(* IEC 61131-3 sources: sphere-usecases/water-treatment/implementations/openplc/projects/controller_project, 4 files *)

(* ---- controller_clean.st ---- *)
TYPE
  HMI_UDT : STRUCT
    Start_PB : BOOL;
    Stop_PB : BOOL;
    Start_Active : BOOL;
    Stop_Active : BOOL;
  END_STRUCT;
  P1_UDT : STRUCT
    RW_Tank_tnk_lvl : REAL;
    RW_Pump_flow : REAL;
    RW_Tank_PR_Valve_sts : BOOL;
    RW_Tank_P6B_Valve_sts : BOOL;
    RW_Tank_P_Valve_sts : BOOL;
    RW_Pump_sts : BOOL;
    RW_Pump_fault : BOOL;
    RW_Pump : REAL;
    RW_Tank_PR_Valve : BOOL;
    RW_Tank_P_Valve : BOOL;
    RW_Pump_start : BOOL;
    RW_Pump_stop : BOOL;
    RW_Tank_P6B_Valve : BOOL;
  END_STRUCT;
  P2_UDT : STRUCT
    ChemTreat_NaCl_Tank_tnk_lvl : REAL;
    ChemTreat_NaOCl_Tank_tnk_lvl : REAL;
    ChemTreat_HCl_Tank_tnk_lvl : REAL;
    ChemTreat_NaCl_Tank_Valve_sts : BOOL;
    ChemTreat_NaOCl_Tank_Valve_sts : BOOL;
    ChemTreat_HCl_Tank_Valve_sts : BOOL;
    ChemTreat_NaCl_Tank_Valve : BOOL;
    ChemTreat_NaOCl_Tank_Valve : BOOL;
    ChemTreat_HCl_Tank_Valve : BOOL;
  END_STRUCT;
  P3_UDT : STRUCT
    Ultrafiltration_UFFT_Tank_tnk_lvl : REAL;
    Ultrafiltration_UFFT_Tank_Valve_sts : BOOL;
    Ultrafiltration_UF_Drain_Valve_sts : BOOL;
    Ultrafiltration_UF_ROFT_Valve_sts : BOOL;
    Ultrafiltration_UF_BWP_Valve_sts : BOOL;
    Ultrafiltration_UFFT_Tank_Valve : BOOL;
    Ultrafiltration_UF_Drain_Valve : BOOL;
    Ultrafiltration_UF_ROFT_Valve : BOOL;
    Ultrafiltration_UF_BWP_Valve : BOOL;
  END_STRUCT;
  Phases_UDT : STRUCT
    Filling : BOOL;
    Draining : BOOL;
  END_STRUCT;
  RW_tank_AL_UDT : STRUCT
    LL_alarm : BOOL;
    L_alarm : BOOL;
    H_alarm : BOOL;
    HH_alarm : BOOL;
  END_STRUCT;
  System_State_UDT : STRUCT
    IDLE : BOOL;
    START : BOOL;
    RUNNING : BOOL;
    SHUTDOWN : BOOL;
    Permissives : ARRAY [0..31] OF BOOL;
    Permissives_Ready : BOOL;
  END_STRUCT;
  SYS_MESSAGES : STRUCT
    ProgramScanTime : DINT;
    AvailableMemory : REAL;
    ControllerStatus : SINT;
    ScanTime : REAL;
  END_STRUCT;
END_TYPE

PROGRAM MainProgram
  VAR_INPUT
    Alarms : RW_tank_AL_UDT;
    GSV_Message : SYS_MESSAGES;
    P1 : P1_UDT;
    P1_SYS : System_State_UDT;
    P2 : P2_UDT;
    P3 : P3_UDT;
  END_VAR
  VAR_INPUT
    di_2_0 AT %IX2.0 : BOOL;
    di_2_1 AT %IX2.1 : BOOL;
    di_2_10 AT %IX2.10 : BOOL;
    di_2_11 AT %IX2.11 : BOOL;
    di_2_2 AT %IX2.2 : BOOL;
    di_2_3 AT %IX2.3 : BOOL;
    di_2_4 AT %IX2.4 : BOOL;
    di_2_5 AT %IX2.5 : BOOL;
    di_2_6 AT %IX2.6 : BOOL;
    di_2_8 AT %IX2.8 : BOOL;
    di_2_9 AT %IX2.9 : BOOL;
    ai_7_0 AT %IW70 : REAL;
    di_7_ch0halarm AT %IX7.0 : BOOL;
    di_7_ch0hhalarm AT %IX7.0 : BOOL;
    di_7_ch0lalarm AT %IX7.0 : BOOL;
    di_7_ch0llalarm AT %IX7.0 : BOOL;
    ai_7_1 AT %IW71 : REAL;
    ai_7_2 AT %IW72 : REAL;
    ai_7_3 AT %IW73 : REAL;
    ai_7_4 AT %IW74 : REAL;
    ai_7_5 AT %IW75 : REAL;
  END_VAR
  VAR_OUTPUT
    HMI : HMI_UDT;
  END_VAR
  VAR_OUTPUT
    ao_10_0 AT %QW100 : REAL;
    do_5_0 AT %QX5.0 : BOOL;
    do_5_1 AT %QX5.1 : BOOL;
    do_5_10 AT %QX5.10 : BOOL;
    do_5_11 AT %QX5.11 : BOOL;
    do_5_2 AT %QX5.2 : BOOL;
    do_5_3 AT %QX5.3 : BOOL;
    do_5_4 AT %QX5.4 : BOOL;
    do_5_5 AT %QX5.5 : BOOL;
    do_5_6 AT %QX5.6 : BOOL;
    do_5_7 AT %QX5.7 : BOOL;
    do_5_8 AT %QX5.8 : BOOL;
    do_5_9 AT %QX5.9 : BOOL;
  END_VAR

  (* IO_setup *)
  (* P1 Analog Input *)
  P1.RW_Tank_tnk_lvl := ai_7_0;
  P1.RW_Pump_flow := ai_7_1;
  (* P1 Digital Input *)
  P1.RW_Tank_PR_Valve_sts := di_2_0;
  P1.RW_Tank_P6B_Valve_sts := di_2_1;
  P1.RW_Tank_P_Valve_sts := di_2_2;
  P1.RW_Pump_sts := di_2_3;
  P1.RW_Pump_fault := di_2_4;
  (* P1 Analog Output *)
  P1.RW_Pump := ao_10_0;
  (* Digital Output *)
  P1.RW_Tank_PR_Valve := do_5_0;
  P1.RW_Tank_P6B_Valve := do_5_1;
  P1.RW_Tank_P_Valve := do_5_2;
  P1.RW_Pump_start := do_5_3;
  P1.RW_Pump_stop := do_5_4;
  (* P1 raw water tank alarms *)
  Alarms.LL_alarm := di_7_ch0llalarm;
  Alarms.L_alarm := di_7_ch0lalarm;
  Alarms.H_alarm := di_7_ch0halarm;
  Alarms.HH_alarm := di_7_ch0hhalarm;
  (* P2 Analog Input *)
  P2.ChemTreat_NaCl_Tank_tnk_lvl := ai_7_2;
  P2.ChemTreat_NaOCl_Tank_tnk_lvl := ai_7_3;
  P2.ChemTreat_HCl_Tank_tnk_lvl := ai_7_4;
  (* P2 Digital Input *)
  P2.ChemTreat_NaCl_Tank_Valve_sts := di_2_5;
  P2.ChemTreat_NaOCl_Tank_Valve_sts := di_2_6;
  (* P2 Analog Output *)
  (* NONE *)
  (* P2 Digital Output *)
  P2.ChemTreat_NaCl_Tank_Valve := do_5_5;
  P2.ChemTreat_NaOCl_Tank_Valve := do_5_6;
  P2.ChemTreat_HCl_Tank_Valve := do_5_7;
  (* P3 Analog Input *)
  P3.Ultrafiltration_UFFT_Tank_tnk_lvl := ai_7_5;
  (* P3 Digital Input *)
  P3.Ultrafiltration_UFFT_Tank_Valve_sts := di_2_8;
  P3.Ultrafiltration_UF_Drain_Valve_sts := di_2_9;
  P3.Ultrafiltration_UF_Drain_Valve_sts := di_2_10;
  P3.Ultrafiltration_UF_BWP_Valve_sts := di_2_11;
  (* P3 Analog Output *)
  (* none *)
  (* P3 Digital Output *)
  P3.Ultrafiltration_UFFT_Tank_Valve := do_5_8;
  P3.Ultrafiltration_UF_Drain_Valve := do_5_9;
  P3.Ultrafiltration_UF_ROFT_Valve := do_5_10;
  P3.Ultrafiltration_UF_BWP_Valve := do_5_11;

  (* Raw_water_control *)
  if P1.RW_Tank_tnk_lvl = 250.0 and P1_SYS.RUNNING then
  P1.RW_Pump_stop := True;
  P1.RW_Pump_start := False; (* send the outputs *)
  Alarms.LL_alarm := True;
  (* if the level is at 500 or lower than 500 open the valve *)
  elsif P1.RW_Tank_tnk_lvl <= 500.0 and P1_SYS.RUNNING then
  (* output to turn the valve open *)
  P1.RW_Tank_PR_Valve := True;
  Alarms.L_alarm := True;
  (* if level is at 800 *)
  elsif  P1.RW_Tank_tnk_lvl = 800.0 and P1_SYS.RUNNING then
  P1.RW_Tank_PR_Valve := False; (* close the valve *)
  Alarms.H_alarm := True;
  elsif P1.RW_Tank_tnk_lvl = 1200.0 and P1_SYS.RUNNING then
  Alarms.HH_alarm := True; (* if the tank is higher than or equal to 1200 set the high high alarm *)
  end_if;

  (* Raw_water_pump *)
  if P3.Ultrafiltration_UFFT_Tank_tnk_lvl = 800.0 AND P1_SYS.RUNNING then
  (* start the pump and open the valve from the other tank *)
  P1.RW_Tank_P_Valve := True;
  P1.RW_Pump_start := True;
  P1.RW_Pump_stop := False;
  elsif P3.Ultrafiltration_UFFT_Tank_tnk_lvl = 1000.0 AND P1_SYS.RUNNING then
  (* stop the pump and close the valve *)
  P1.RW_Tank_P_Valve := False;
  P1.RW_Pump_stop := True;
  P1.RW_Pump_start := False;
  end_if;

  (* State_change *)
  if not HMI.Start_Active AND not HMI.Stop_Active then
  (* if start and stop is not pressed go to idle *)
  P1_SYS.IDLE := True;
  P1_SYS.START := False;
  P1_SYS.RUNNING := False;
  P1_SYS.SHUTDOWN := False;
  elsif  HMI.Start_Active AND not HMI.Stop_Active then
  (* if the start pb and stop is not pressed then change the state of process one to starting *)
  P1_SYS.IDLE := False;
  P1_SYS.START := True;
  P1_SYS.RUNNING := False;
  P1_SYS.SHUTDOWN := False;
  (* if the tank level is greater than 250 at the start and UFFT is less than a 1000 we can start *)
  (* then and all permissves cond together into one tag so we know the plant is ready to start *)
  P1_SYS.Permissives_Ready := P1_SYS.Permissives[0] AND P1_SYS.Permissives[1];
  elsif HMI.Start_Active AND P1_SYS.Permissives_Ready then
  (* if the start was pressed and permissives are ready start running Process one *)
  P1_SYS.IDLE := False;
  P1_SYS.START := False;
  P1_SYS.RUNNING := True;
  P1_SYS.SHUTDOWN := False;
  elsif HMI.Stop_Active then
  (* if the stop button is pressed then go to shutdown state *)
  P1_SYS.IDLE := False;
  P1_SYS.START := False;
  P1_SYS.RUNNING := False;
  P1_SYS.SHUTDOWN := True;
  (* set all permissives to false *)
  P1_SYS.Permissives_Ready := False;
  end_if;
END_PROGRAM

CONFIGURATION config
  VAR_GLOBAL
    ao_10_0 AT %QW100 : REAL;
    di_2_0 AT %IX2.0 : BOOL;
    di_2_1 AT %IX2.1 : BOOL;
    di_2_10 AT %IX2.10 : BOOL;
    di_2_11 AT %IX2.11 : BOOL;
    di_2_2 AT %IX2.2 : BOOL;
    di_2_3 AT %IX2.3 : BOOL;
    di_2_4 AT %IX2.4 : BOOL;
    di_2_5 AT %IX2.5 : BOOL;
    di_2_6 AT %IX2.6 : BOOL;
    di_2_8 AT %IX2.8 : BOOL;
    di_2_9 AT %IX2.9 : BOOL;
    do_5_0 AT %QX5.0 : BOOL;
    do_5_1 AT %QX5.1 : BOOL;
    do_5_10 AT %QX5.10 : BOOL;
    do_5_11 AT %QX5.11 : BOOL;
    do_5_2 AT %QX5.2 : BOOL;
    do_5_3 AT %QX5.3 : BOOL;
    do_5_4 AT %QX5.4 : BOOL;
    do_5_5 AT %QX5.5 : BOOL;
    do_5_6 AT %QX5.6 : BOOL;
    do_5_7 AT %QX5.7 : BOOL;
    do_5_8 AT %QX5.8 : BOOL;
    do_5_9 AT %QX5.9 : BOOL;
    ai_7_0 AT %IW70 : REAL;
    di_7_ch0halarm AT %IX7.0 : BOOL;
    di_7_ch0hhalarm AT %IX7.0 : BOOL;
    di_7_ch0lalarm AT %IX7.0 : BOOL;
    di_7_ch0llalarm AT %IX7.0 : BOOL;
    ai_7_1 AT %IW71 : REAL;
    ai_7_2 AT %IW72 : REAL;
    ai_7_3 AT %IW73 : REAL;
    ai_7_4 AT %IW74 : REAL;
    ai_7_5 AT %IW75 : REAL;
  END_VAR

  RESOURCE res_MainProgram ON PLC
    TASK task_MainProgram(INTERVAL := T#100ms,PRIORITY := 0);
    PROGRAM MainProgram_instance : MainProgram;
  END_RESOURCE
END_CONFIGURATION

(* ---- controller_final.st ---- *)
TYPE
  HMI_UDT : STRUCT
    Start_PB : BOOL;
    Stop_PB : BOOL;
    Reset_PB : BOOL;
    Start_Active : BOOL;
    Stop_Active : BOOL;
  END_STRUCT;
  P1_UDT : STRUCT
    RW_Tank_tnk_lvl : REAL;
    RW_Pump_flow : REAL;
    RW_Tank_PR_Valve_sts : BOOL;
    RW_Tank_P6B_Valve_sts : BOOL;
    RW_Tank_P_Valve_sts : BOOL;
    RW_Pump_sts : BOOL;
    RW_Pump_fault : BOOL;
    RW_Pump : REAL;
    RW_Tank_PR_Valve : BOOL;
    RW_Tank_P_Valve : BOOL;
    RW_Pump_start : BOOL;
    RW_Pump_stop : BOOL;
    RW_Tank_P6B_Valve : BOOL;
  END_STRUCT;
  P2_UDT : STRUCT
    ChemTreat_NaCl_Tank_tnk_lvl : REAL;
    ChemTreat_NaOCl_Tank_tnk_lvl : REAL;
    ChemTreat_HCl_Tank_tnk_lvl : REAL;
    ChemTreat_NaCl_Tank_Valve_sts : BOOL;
    ChemTreat_NaOCl_Tank_Valve_sts : BOOL;
    ChemTreat_HCl_Tank_Valve_sts : BOOL;
    ChemTreat_NaCl_Tank_Valve : BOOL;
    ChemTreat_NaOCl_Tank_Valve : BOOL;
    ChemTreat_HCl_Tank_Valve : BOOL;
  END_STRUCT;
  P3_UDT : STRUCT
    Ultrafiltration_UFFT_Tank_tnk_lvl : REAL;
    Ultrafiltration_UFFT_Tank_Valve_sts : BOOL;
    Ultrafiltration_UF_Drain_Valve_sts : BOOL;
    Ultrafiltration_UF_ROFT_Valve_sts : BOOL;
    Ultrafiltration_UF_BWP_Valve_sts : BOOL;
    Ultrafiltration_UFFT_Tank_Valve : BOOL;
    Ultrafiltration_UF_Drain_Valve : BOOL;
    Ultrafiltration_UF_ROFT_Valve : BOOL;
    Ultrafiltration_UF_BWP_Valve : BOOL;
  END_STRUCT;
  Phases_UDT : STRUCT
    Filling : BOOL;
    Draining : BOOL;
  END_STRUCT;
  RW_tank_AL_UDT : STRUCT
    LL_alarm : BOOL;
    L_alarm : BOOL;
    H_alarm : BOOL;
    HH_alarm : BOOL;
  END_STRUCT;
  System_State_UDT : STRUCT
    IDLE : BOOL;
    START : BOOL;
    RUNNING : BOOL;
    SHUTDOWN : BOOL;
    Permissives : ARRAY [0..31] OF BOOL;
    Permissives_Ready : BOOL;
  END_STRUCT;
  SYS_MESSAGES : STRUCT
    ProgramScanTime : DINT;
    AvailableMemory : REAL;
    ControllerStatus : SINT;
    ScanTime : REAL;
  END_STRUCT;
END_TYPE

PROGRAM MainProgram
  VAR
    HMI : HMI_UDT;
    Alarms : RW_tank_AL_UDT;
    GSV_Message : SYS_MESSAGES;
    Init_Done : BOOL := FALSE;
    P1 : P1_UDT;
    P1_SYS : System_State_UDT;
    P2 : P2_UDT;
    P3 : P3_UDT;
  END_VAR
  VAR_EXTERNAL
    ao_10_0 : INT;
    do_5_0 : BOOL;
    do_5_1 : BOOL;
    do_5_10 : BOOL;
    do_5_11 : BOOL;
    do_5_2 : BOOL;
    do_5_3 : BOOL;
    do_5_4 : BOOL;
    do_5_5 : BOOL;
    do_5_6 : BOOL;
    do_5_7 : BOOL;
    do_5_8 : BOOL;
    do_5_9 : BOOL;
    (* HMI coils %QX0.0-0.3 *)
    hmi_0_0 : BOOL;  (* HMI_Start_PB - written by external client *)
    hmi_0_1 : BOOL;  (* HMI_Stop_PB  - written by external client *)
    hmi_0_2 : BOOL;  (* HMI_Start_Active - written by controller *)
    hmi_0_3 : BOOL;  (* HMI_Stop_Active  - written by controller *)
    hmi_0_4 : BOOL;  (* HMI_Reset_PB - written by external client *)
    (* Process selection/manual P2 control coils %QX1.0-1.3 *)
    p2_1_0 : BOOL;  (* P2_Selected - written by external client *)
    p2_1_1 : BOOL;  (* P2_NaCl_Cmd - written by external client *)
    p2_1_2 : BOOL;  (* P2_NaOCl_Cmd - written by external client *)
    p2_1_3 : BOOL;  (* P2_HCl_Cmd - written by external client *)
    (* System state coils %QX7.0-7.4 *)
    sys_7_0 : BOOL;  (* SYS_IDLE *)
    sys_7_1 : BOOL;  (* SYS_START *)
    sys_7_2 : BOOL;  (* SYS_RUNNING *)
    sys_7_3 : BOOL;  (* SYS_SHUTDOWN *)
    sys_7_4 : BOOL;  (* SYS_Permissives_Ready *)
    (* Alarm coils %QX8.0-8.3 *)
    alm_8_0 : BOOL;  (* Alarm_RW_Tank_LL *)
    alm_8_1 : BOOL;  (* Alarm_RW_Tank_L *)
    alm_8_2 : BOOL;  (* Alarm_RW_Tank_H *)
    alm_8_3 : BOOL;  (* Alarm_RW_Tank_HH *)
    (* Bridge sensor inputs - holding registers written by bridge *)
    bridge_rw_level : INT;       (* %QW300 - RW tank level from simulator *)
    bridge_rw_flow : INT;        (* %QW301 - RW pump flow from simulator *)
    bridge_nacl_level : INT;     (* %QW302 - NaCl tank level *)
    bridge_naocl_level : INT;    (* %QW303 - NaOCl tank level *)
    bridge_hcl_level : INT;      (* %QW304 - HCl tank level *)
    bridge_uf_level : INT;       (* %QW305 - UF tank level *)
    bridge_pr_valve_sts : INT;   (* %QW320 - PR valve status *)
    bridge_p6b_valve_sts : INT;  (* %QW321 - P6B valve status *)
    bridge_p_valve_sts : INT;    (* %QW322 - P valve status *)
    bridge_pump_sts : INT;       (* %QW323 - pump running status *)
    bridge_pump_fault : INT;     (* %QW324 - pump fault *)
    bridge_nacl_valve_sts : INT; (* %QW325 - NaCl valve status *)
    bridge_naocl_valve_sts : INT;(* %QW326 - NaOCl valve status *)
    bridge_hcl_valve_sts : INT;  (* %QW327 - HCl valve status *)
    bridge_uf_valve_sts : INT;   (* %QW328 - UF tank valve status *)
    bridge_uf_drain_sts : INT;   (* %QW329 - UF drain valve status *)
    bridge_uf_roft_sts : INT;    (* %QW330 - UF ROFT valve status *)
    bridge_uf_bwp_sts : INT;     (* %QW331 - UF BWP valve status *)
  END_VAR

  IF NOT Init_Done THEN
    HMI.Start_Active := FALSE;
    HMI.Stop_Active := FALSE;
    P1_SYS.IDLE := TRUE;
    P1_SYS.START := FALSE;
    P1_SYS.RUNNING := FALSE;
    P1_SYS.SHUTDOWN := FALSE;
    P1_SYS.Permissives_Ready := FALSE;
    P1.RW_Pump := 0.0;
    P1.RW_Tank_PR_Valve := FALSE;
    P1.RW_Tank_P_Valve := FALSE;
    P1.RW_Pump_start := FALSE;
    P1.RW_Pump_stop := TRUE;
    P1.RW_Tank_P6B_Valve := FALSE;
    P2.ChemTreat_NaCl_Tank_Valve := FALSE;
    P2.ChemTreat_NaOCl_Tank_Valve := FALSE;
    P2.ChemTreat_HCl_Tank_Valve := FALSE;
    P3.Ultrafiltration_UFFT_Tank_Valve := FALSE;
    P3.Ultrafiltration_UF_Drain_Valve := FALSE;
    P3.Ultrafiltration_UF_ROFT_Valve := FALSE;
    P3.Ultrafiltration_UF_BWP_Valve := FALSE;
    Init_Done := TRUE;
  END_IF;

  (* ===== HMI button latch ===== *)
  HMI.Start_PB := hmi_0_0;
  HMI.Stop_PB := hmi_0_1;
  HMI.Reset_PB := hmi_0_4;
  IF HMI.Reset_PB THEN
    HMI.Start_Active := FALSE;
    HMI.Stop_Active := FALSE;
  ELSIF HMI.Start_PB THEN
    HMI.Start_Active := TRUE;
    HMI.Stop_Active := FALSE;
  ELSIF HMI.Stop_PB THEN
    HMI.Stop_Active := TRUE;
    HMI.Start_Active := FALSE;
  END_IF;

  (* ===== Read sensors from bridge holding registers ===== *)
  (* Levels: INT -> REAL conversion *)
  P1.RW_Tank_tnk_lvl := INT_TO_REAL(bridge_rw_level);
  P1.RW_Pump_flow := INT_TO_REAL(bridge_rw_flow);
  P2.ChemTreat_NaCl_Tank_tnk_lvl := INT_TO_REAL(bridge_nacl_level);
  P2.ChemTreat_NaOCl_Tank_tnk_lvl := INT_TO_REAL(bridge_naocl_level);
  P2.ChemTreat_HCl_Tank_tnk_lvl := INT_TO_REAL(bridge_hcl_level);
  P3.Ultrafiltration_UFFT_Tank_tnk_lvl := INT_TO_REAL(bridge_uf_level);
  (* Valve/pump status: INT -> BOOL (nonzero = TRUE) *)
  P1.RW_Tank_PR_Valve_sts := bridge_pr_valve_sts <> 0;
  P1.RW_Tank_P6B_Valve_sts := bridge_p6b_valve_sts <> 0;
  P1.RW_Tank_P_Valve_sts := bridge_p_valve_sts <> 0;
  P1.RW_Pump_sts := bridge_pump_sts <> 0;
  P1.RW_Pump_fault := bridge_pump_fault <> 0;
  P2.ChemTreat_NaCl_Tank_Valve_sts := bridge_nacl_valve_sts <> 0;
  P2.ChemTreat_NaOCl_Tank_Valve_sts := bridge_naocl_valve_sts <> 0;
  P3.Ultrafiltration_UFFT_Tank_Valve_sts := bridge_uf_valve_sts <> 0;
  P3.Ultrafiltration_UF_Drain_Valve_sts := bridge_uf_drain_sts <> 0;
  P3.Ultrafiltration_UF_ROFT_Valve_sts := bridge_uf_roft_sts <> 0;
  P3.Ultrafiltration_UF_BWP_Valve_sts := bridge_uf_bwp_sts <> 0;

  (* ===== Compute alarms from levels ===== *)
  Alarms.LL_alarm := P1.RW_Tank_tnk_lvl <= 250.0;
  Alarms.L_alarm := P1.RW_Tank_tnk_lvl <= 500.0;
  Alarms.H_alarm := P1.RW_Tank_tnk_lvl >= 800.0;
  Alarms.HH_alarm := P1.RW_Tank_tnk_lvl >= 1200.0;

  (* ===== Permissives ===== *)
  P1_SYS.Permissives[0] := P1.RW_Tank_tnk_lvl > 250.0;
  P1_SYS.Permissives[1] := P3.Ultrafiltration_UFFT_Tank_tnk_lvl < 1000.0;
  P1_SYS.Permissives_Ready := P1_SYS.Permissives[0] AND P1_SYS.Permissives[1];

  (* ===== State_change ===== *)
  IF HMI.Reset_PB THEN
    P1_SYS.IDLE := TRUE;
    P1_SYS.START := FALSE;
    P1_SYS.RUNNING := FALSE;
    P1_SYS.SHUTDOWN := FALSE;
    P1_SYS.Permissives_Ready := FALSE;
    P1.RW_Pump := 0.0;
    P1.RW_Tank_PR_Valve := FALSE;
    P1.RW_Tank_P_Valve := FALSE;
    P1.RW_Pump_start := FALSE;
    P1.RW_Pump_stop := TRUE;
  ELSIF NOT HMI.Start_Active AND NOT HMI.Stop_Active THEN
    P1_SYS.IDLE := TRUE;
    P1_SYS.START := FALSE;
    P1_SYS.RUNNING := FALSE;
    P1_SYS.SHUTDOWN := FALSE;
    P1_SYS.Permissives_Ready := FALSE;
    P1.RW_Pump := 0.0;
    P1.RW_Tank_PR_Valve := FALSE;
    P1.RW_Tank_P_Valve := FALSE;
    P1.RW_Pump_start := FALSE;
    P1.RW_Pump_stop := TRUE;
  ELSIF HMI.Start_Active AND NOT HMI.Stop_Active AND NOT P1_SYS.Permissives_Ready THEN
    P1_SYS.IDLE := FALSE;
    P1_SYS.START := TRUE;
    P1_SYS.RUNNING := FALSE;
    P1_SYS.SHUTDOWN := FALSE;
  ELSIF HMI.Start_Active AND P1_SYS.Permissives_Ready THEN
    P1_SYS.IDLE := FALSE;
    P1_SYS.START := FALSE;
    P1_SYS.RUNNING := TRUE;
    P1_SYS.SHUTDOWN := FALSE;
  ELSIF HMI.Stop_Active THEN
    P1_SYS.IDLE := FALSE;
    P1_SYS.START := FALSE;
    P1_SYS.RUNNING := FALSE;
    P1_SYS.SHUTDOWN := TRUE;
    P1_SYS.Permissives_Ready := FALSE;
    P1.RW_Pump := 0.0;
    P1.RW_Tank_PR_Valve := FALSE;
    P1.RW_Tank_P_Valve := FALSE;
    P1.RW_Pump_start := FALSE;
    P1.RW_Pump_stop := TRUE;
  END_IF;

  (* ===== Raw_water_control ===== *)
  IF P1_SYS.RUNNING THEN
    IF P1.RW_Tank_tnk_lvl <= 250.0 THEN
      P1.RW_Pump_stop := TRUE;
      P1.RW_Pump_start := FALSE;
      P1.RW_Tank_P_Valve := FALSE;
      P1.RW_Pump := 0.0;
    ELSIF P1.RW_Tank_tnk_lvl <= 500.0 THEN
      P1.RW_Tank_PR_Valve := TRUE;
    ELSIF P1.RW_Tank_tnk_lvl >= 800.0 THEN
      P1.RW_Tank_PR_Valve := FALSE;
    END_IF;

    (* ===== Raw_water_pump ===== *)
    IF P3.Ultrafiltration_UFFT_Tank_tnk_lvl <= 800.0 THEN
      P1.RW_Tank_P_Valve := TRUE;
      P1.RW_Pump_start := TRUE;
      P1.RW_Pump_stop := FALSE;
      P1.RW_Pump := 100.0;
    ELSIF P3.Ultrafiltration_UFFT_Tank_tnk_lvl >= 1000.0 THEN
      P1.RW_Tank_P_Valve := FALSE;
      P1.RW_Pump_stop := TRUE;
      P1.RW_Pump_start := FALSE;
      P1.RW_Pump := 0.0;
    END_IF;
  END_IF;

  (* ===== Manual Process 2 control ===== *)
  IF P1_SYS.RUNNING AND p2_1_0 THEN
    P2.ChemTreat_NaCl_Tank_Valve := p2_1_1;
    P2.ChemTreat_NaOCl_Tank_Valve := p2_1_2;
    P2.ChemTreat_HCl_Tank_Valve := p2_1_3;
  ELSE
    P2.ChemTreat_NaCl_Tank_Valve := FALSE;
    P2.ChemTreat_NaOCl_Tank_Valve := FALSE;
    P2.ChemTreat_HCl_Tank_Valve := FALSE;
  END_IF;

  (* ===== Wire outputs to coils/registers ===== *)
  do_5_0 := P1.RW_Tank_PR_Valve;
  do_5_1 := P1.RW_Tank_P6B_Valve;
  do_5_2 := P1.RW_Tank_P_Valve;
  do_5_3 := P1.RW_Pump_start;
  do_5_4 := P1.RW_Pump_stop;
  do_5_5 := P2.ChemTreat_NaCl_Tank_Valve;
  do_5_6 := P2.ChemTreat_NaOCl_Tank_Valve;
  do_5_7 := P2.ChemTreat_HCl_Tank_Valve;
  do_5_8 := P3.Ultrafiltration_UFFT_Tank_Valve;
  do_5_9 := P3.Ultrafiltration_UF_Drain_Valve;
  do_5_10 := P3.Ultrafiltration_UF_ROFT_Valve;
  do_5_11 := P3.Ultrafiltration_UF_BWP_Valve;
  ao_10_0 := REAL_TO_INT(P1.RW_Pump);
  (* HMI status *)
  hmi_0_2 := HMI.Start_Active;
  hmi_0_3 := HMI.Stop_Active;
  (* System state *)
  sys_7_0 := P1_SYS.IDLE;
  sys_7_1 := P1_SYS.START;
  sys_7_2 := P1_SYS.RUNNING;
  sys_7_3 := P1_SYS.SHUTDOWN;
  sys_7_4 := P1_SYS.Permissives_Ready;
  (* Alarms *)
  alm_8_0 := Alarms.LL_alarm;
  alm_8_1 := Alarms.L_alarm;
  alm_8_2 := Alarms.H_alarm;
  alm_8_3 := Alarms.HH_alarm;
END_PROGRAM

CONFIGURATION Config0
  VAR_GLOBAL
    ao_10_0 AT %QW100 : INT;
    do_5_0 AT %QX5.0 : BOOL;
    do_5_1 AT %QX5.1 : BOOL;
    do_5_10 AT %QX5.10 : BOOL;
    do_5_11 AT %QX5.11 : BOOL;
    do_5_2 AT %QX5.2 : BOOL;
    do_5_3 AT %QX5.3 : BOOL;
    do_5_4 AT %QX5.4 : BOOL;
    do_5_5 AT %QX5.5 : BOOL;
    do_5_6 AT %QX5.6 : BOOL;
    do_5_7 AT %QX5.7 : BOOL;
    do_5_8 AT %QX5.8 : BOOL;
    do_5_9 AT %QX5.9 : BOOL;
    (* HMI coils %QX0.0-0.4 *)
    hmi_0_0 AT %QX0.0 : BOOL;
    hmi_0_1 AT %QX0.1 : BOOL;
    hmi_0_2 AT %QX0.2 : BOOL;
    hmi_0_3 AT %QX0.3 : BOOL;
    hmi_0_4 AT %QX0.4 : BOOL;
    (* Process selection/manual P2 control coils %QX1.0-1.3 *)
    p2_1_0 AT %QX1.0 : BOOL;
    p2_1_1 AT %QX1.1 : BOOL;
    p2_1_2 AT %QX1.2 : BOOL;
    p2_1_3 AT %QX1.3 : BOOL;
    (* System state coils %QX7.0-7.4 *)
    sys_7_0 AT %QX7.0 : BOOL;
    sys_7_1 AT %QX7.1 : BOOL;
    sys_7_2 AT %QX7.2 : BOOL;
    sys_7_3 AT %QX7.3 : BOOL;
    sys_7_4 AT %QX7.4 : BOOL;
    (* Alarm coils %QX8.0-8.3 *)
    alm_8_0 AT %QX8.0 : BOOL;
    alm_8_1 AT %QX8.1 : BOOL;
    alm_8_2 AT %QX8.2 : BOOL;
    alm_8_3 AT %QX8.3 : BOOL;
    (* Bridge sensor inputs - holding registers writable by bridge *)
    bridge_rw_level AT %QW300 : INT;
    bridge_rw_flow AT %QW301 : INT;
    bridge_nacl_level AT %QW302 : INT;
    bridge_naocl_level AT %QW303 : INT;
    bridge_hcl_level AT %QW304 : INT;
    bridge_uf_level AT %QW305 : INT;
    bridge_pr_valve_sts AT %QW320 : INT;
    bridge_p6b_valve_sts AT %QW321 : INT;
    bridge_p_valve_sts AT %QW322 : INT;
    bridge_pump_sts AT %QW323 : INT;
    bridge_pump_fault AT %QW324 : INT;
    bridge_nacl_valve_sts AT %QW325 : INT;
    bridge_naocl_valve_sts AT %QW326 : INT;
    bridge_hcl_valve_sts AT %QW327 : INT;
    bridge_uf_valve_sts AT %QW328 : INT;
    bridge_uf_drain_sts AT %QW329 : INT;
    bridge_uf_roft_sts AT %QW330 : INT;
    bridge_uf_bwp_sts AT %QW331 : INT;
  END_VAR

  RESOURCE Res0 ON PLC
    TASK task_MainProgram(INTERVAL := T#100ms, PRIORITY := 0);
    PROGRAM MainProgram_instance : MainProgram;
  END_RESOURCE
END_CONFIGURATION

(* ---- controller_fixed.st ---- *)
TYPE
  HMI_UDT : STRUCT
    Start_PB : BOOL;
    Stop_PB : BOOL;
    Start_Active : BOOL;
    Stop_Active : BOOL;
  END_STRUCT;
  P1_UDT : STRUCT
    RW_Tank_tnk_lvl : REAL;
    RW_Pump_flow : REAL;
    RW_Tank_PR_Valve_sts : BOOL;
    RW_Tank_P6B_Valve_sts : BOOL;
    RW_Tank_P_Valve_sts : BOOL;
    RW_Pump_sts : BOOL;
    RW_Pump_fault : BOOL;
    RW_Pump : REAL;
    RW_Tank_PR_Valve : BOOL;
    RW_Tank_P_Valve : BOOL;
    RW_Pump_start : BOOL;
    RW_Pump_stop : BOOL;
    RW_Tank_P6B_Valve : BOOL;
  END_STRUCT;
  P2_UDT : STRUCT
    ChemTreat_NaCl_Tank_tnk_lvl : REAL;
    ChemTreat_NaOCl_Tank_tnk_lvl : REAL;
    ChemTreat_HCl_Tank_tnk_lvl : REAL;
    ChemTreat_NaCl_Tank_Valve_sts : BOOL;
    ChemTreat_NaOCl_Tank_Valve_sts : BOOL;
    ChemTreat_HCl_Tank_Valve_sts : BOOL;
    ChemTreat_NaCl_Tank_Valve : BOOL;
    ChemTreat_NaOCl_Tank_Valve : BOOL;
    ChemTreat_HCl_Tank_Valve : BOOL;
  END_STRUCT;
  P3_UDT : STRUCT
    Ultrafiltration_UFFT_Tank_tnk_lvl : REAL;
    Ultrafiltration_UFFT_Tank_Valve_sts : BOOL;
    Ultrafiltration_UF_Drain_Valve_sts : BOOL;
    Ultrafiltration_UF_ROFT_Valve_sts : BOOL;
    Ultrafiltration_UF_BWP_Valve_sts : BOOL;
    Ultrafiltration_UFFT_Tank_Valve : BOOL;
    Ultrafiltration_UF_Drain_Valve : BOOL;
    Ultrafiltration_UF_ROFT_Valve : BOOL;
    Ultrafiltration_UF_BWP_Valve : BOOL;
  END_STRUCT;
  Phases_UDT : STRUCT
    Filling : BOOL;
    Draining : BOOL;
  END_STRUCT;
  RW_tank_AL_UDT : STRUCT
    LL_alarm : BOOL;
    L_alarm : BOOL;
    H_alarm : BOOL;
    HH_alarm : BOOL;
  END_STRUCT;
  System_State_UDT : STRUCT
    IDLE : BOOL;
    START : BOOL;
    RUNNING : BOOL;
    SHUTDOWN : BOOL;
    Permissives : ARRAY [0..31] OF BOOL;
    Permissives_Ready : BOOL;
  END_STRUCT;
  SYS_MESSAGES : STRUCT
    ProgramScanTime : DINT;
    AvailableMemory : REAL;
    ControllerStatus : SINT;
    ScanTime : REAL;
  END_STRUCT;
END_TYPE

PROGRAM MainProgram
  VAR_INPUT
    Alarms : RW_tank_AL_UDT;
    GSV_Message : SYS_MESSAGES;
    P1 : P1_UDT;
    P1_SYS : System_State_UDT;
    P2 : P2_UDT;
    P3 : P3_UDT;
  END_VAR
  VAR_INPUT
    di_2_0 : BOOL;
    di_2_1 : BOOL;
    di_2_10 : BOOL;
    di_2_11 : BOOL;
    di_2_2 : BOOL;
    di_2_3 : BOOL;
    di_2_4 : BOOL;
    di_2_5 : BOOL;
    di_2_6 : BOOL;
    di_2_8 : BOOL;
    di_2_9 : BOOL;
    ai_7_0 : REAL;
    di_7_ch0halarm : BOOL;
    di_7_ch0hhalarm : BOOL;
    di_7_ch0lalarm : BOOL;
    di_7_ch0llalarm : BOOL;
    ai_7_1 : REAL;
    ai_7_2 : REAL;
    ai_7_3 : REAL;
    ai_7_4 : REAL;
    ai_7_5 : REAL;
  END_VAR
  VAR_OUTPUT
    HMI : HMI_UDT;
  END_VAR
  VAR_OUTPUT
    ao_10_0 : REAL;
    do_5_0 : BOOL;
    do_5_1 : BOOL;
    do_5_10 : BOOL;
    do_5_11 : BOOL;
    do_5_2 : BOOL;
    do_5_3 : BOOL;
    do_5_4 : BOOL;
    do_5_5 : BOOL;
    do_5_6 : BOOL;
    do_5_7 : BOOL;
    do_5_8 : BOOL;
    do_5_9 : BOOL;
  END_VAR

  (* IO_setup *)
  (* P1 Analog Input *)
  P1.RW_Tank_tnk_lvl := ai_7_0;
  P1.RW_Pump_flow := ai_7_1;
  (* P1 Digital Input *)
  P1.RW_Tank_PR_Valve_sts := di_2_0;
  P1.RW_Tank_P6B_Valve_sts := di_2_1;
  P1.RW_Tank_P_Valve_sts := di_2_2;
  P1.RW_Pump_sts := di_2_3;
  P1.RW_Pump_fault := di_2_4;
  (* P1 Analog Output *)
  P1.RW_Pump := ao_10_0;
  (* Digital Output *)
  P1.RW_Tank_PR_Valve := do_5_0;
  P1.RW_Tank_P6B_Valve := do_5_1;
  P1.RW_Tank_P_Valve := do_5_2;
  P1.RW_Pump_start := do_5_3;
  P1.RW_Pump_stop := do_5_4;
  (* P1 raw water tank alarms *)
  Alarms.LL_alarm := di_7_ch0llalarm;
  Alarms.L_alarm := di_7_ch0lalarm;
  Alarms.H_alarm := di_7_ch0halarm;
  Alarms.HH_alarm := di_7_ch0hhalarm;
  (* P2 Analog Input *)
  P2.ChemTreat_NaCl_Tank_tnk_lvl := ai_7_2;
  P2.ChemTreat_NaOCl_Tank_tnk_lvl := ai_7_3;
  P2.ChemTreat_HCl_Tank_tnk_lvl := ai_7_4;
  (* P2 Digital Input *)
  P2.ChemTreat_NaCl_Tank_Valve_sts := di_2_5;
  P2.ChemTreat_NaOCl_Tank_Valve_sts := di_2_6;
  (* P2 Analog Output *)
  (* NONE *)
  (* P2 Digital Output *)
  P2.ChemTreat_NaCl_Tank_Valve := do_5_5;
  P2.ChemTreat_NaOCl_Tank_Valve := do_5_6;
  P2.ChemTreat_HCl_Tank_Valve := do_5_7;
  (* P3 Analog Input *)
  P3.Ultrafiltration_UFFT_Tank_tnk_lvl := ai_7_5;
  (* P3 Digital Input *)
  P3.Ultrafiltration_UFFT_Tank_Valve_sts := di_2_8;
  P3.Ultrafiltration_UF_Drain_Valve_sts := di_2_9;
  P3.Ultrafiltration_UF_Drain_Valve_sts := di_2_10;
  P3.Ultrafiltration_UF_BWP_Valve_sts := di_2_11;
  (* P3 Analog Output *)
  (* none *)
  (* P3 Digital Output *)
  P3.Ultrafiltration_UFFT_Tank_Valve := do_5_8;
  P3.Ultrafiltration_UF_Drain_Valve := do_5_9;
  P3.Ultrafiltration_UF_ROFT_Valve := do_5_10;
  P3.Ultrafiltration_UF_BWP_Valve := do_5_11;

  (* Raw_water_control *)
  if P1.RW_Tank_tnk_lvl = 250.0 and P1_SYS.RUNNING then
  P1.RW_Pump_stop := True;
  P1.RW_Pump_start := False; (* send the outputs *)
  Alarms.LL_alarm := True;
  (* if the level is at 500 or lower than 500 open the valve *)
  elsif P1.RW_Tank_tnk_lvl <= 500.0 and P1_SYS.RUNNING then
  (* output to turn the valve open *)
  P1.RW_Tank_PR_Valve := True;
  Alarms.L_alarm := True;
  (* if level is at 800 *)
  elsif  P1.RW_Tank_tnk_lvl = 800.0 and P1_SYS.RUNNING then
  P1.RW_Tank_PR_Valve := False; (* close the valve *)
  Alarms.H_alarm := True;
  elsif P1.RW_Tank_tnk_lvl = 1200.0 and P1_SYS.RUNNING then
  Alarms.HH_alarm := True; (* if the tank is higher than or equal to 1200 set the high high alarm *)
  end_if;

  (* Raw_water_pump *)
  if P3.Ultrafiltration_UFFT_Tank_tnk_lvl = 800.0 AND P1_SYS.RUNNING then
  (* start the pump and open the valve from the other tank *)
  P1.RW_Tank_P_Valve := True;
  P1.RW_Pump_start := True;
  P1.RW_Pump_stop := False;
  elsif P3.Ultrafiltration_UFFT_Tank_tnk_lvl = 1000.0 AND P1_SYS.RUNNING then
  (* stop the pump and close the valve *)
  P1.RW_Tank_P_Valve := False;
  P1.RW_Pump_stop := True;
  P1.RW_Pump_start := False;
  end_if;

  (* State_change *)
  if not HMI.Start_Active AND not HMI.Stop_Active then
  (* if start and stop is not pressed go to idle *)
  P1_SYS.IDLE := True;
  P1_SYS.START := False;
  P1_SYS.RUNNING := False;
  P1_SYS.SHUTDOWN := False;
  elsif  HMI.Start_Active AND not HMI.Stop_Active then
  (* if the start pb and stop is not pressed then change the state of process one to starting *)
  P1_SYS.IDLE := False;
  P1_SYS.START := True;
  P1_SYS.RUNNING := False;
  P1_SYS.SHUTDOWN := False;
  (* if the tank level is greater than 250 at the start and UFFT is less than a 1000 we can start *)
  (* then and all permissves cond together into one tag so we know the plant is ready to start *)
  P1_SYS.Permissives_Ready := P1_SYS.Permissives[0] AND P1_SYS.Permissives[1];
  elsif HMI.Start_Active AND P1_SYS.Permissives_Ready then
  (* if the start was pressed and permissives are ready start running Process one *)
  P1_SYS.IDLE := False;
  P1_SYS.START := False;
  P1_SYS.RUNNING := True;
  P1_SYS.SHUTDOWN := False;
  elsif HMI.Stop_Active then
  (* if the stop button is pressed then go to shutdown state *)
  P1_SYS.IDLE := False;
  P1_SYS.START := False;
  P1_SYS.RUNNING := False;
  P1_SYS.SHUTDOWN := True;
  (* set all permissives to false *)
  P1_SYS.Permissives_Ready := False;
  end_if;
END_PROGRAM

CONFIGURATION config
  VAR_GLOBAL
    ao_10_0 : REAL;
    di_2_0 : BOOL;
    di_2_1 : BOOL;
    di_2_10 : BOOL;
    di_2_11 : BOOL;
    di_2_2 : BOOL;
    di_2_3 : BOOL;
    di_2_4 : BOOL;
    di_2_5 : BOOL;
    di_2_6 : BOOL;
    di_2_8 : BOOL;
    di_2_9 : BOOL;
    do_5_0 : BOOL;
    do_5_1 : BOOL;
    do_5_10 : BOOL;
    do_5_11 : BOOL;
    do_5_2 : BOOL;
    do_5_3 : BOOL;
    do_5_4 : BOOL;
    do_5_5 : BOOL;
    do_5_6 : BOOL;
    do_5_7 : BOOL;
    do_5_8 : BOOL;
    do_5_9 : BOOL;
    ai_7_0 : REAL;
    di_7_ch0halarm : BOOL;
    di_7_ch0hhalarm : BOOL;
    di_7_ch0lalarm : BOOL;
    di_7_ch0llalarm : BOOL;
    ai_7_1 : REAL;
    ai_7_2 : REAL;
    ai_7_3 : REAL;
    ai_7_4 : REAL;
    ai_7_5 : REAL;
  END_VAR

  RESOURCE res_MainProgram ON PLC
    TASK task_MainProgram(INTERVAL := T#100ms,PRIORITY := 0);
    PROGRAM MainProgram_instance : MainProgram;
  END_RESOURCE
END_CONFIGURATION

(* ---- controller_st_file_to_upload.st ---- *)
TYPE
  HMI_UDT : STRUCT
    Start_PB : BOOL;
    Stop_PB : BOOL;
    Start_Active : BOOL;
    Stop_Active : BOOL;
  END_STRUCT;
  P1_UDT : STRUCT
    RW_Tank_tnk_lvl : REAL;
    RW_Pump_flow : REAL;
    RW_Tank_PR_Valve_sts : BOOL;
    RW_Tank_P6B_Valve_sts : BOOL;
    RW_Tank_P_Valve_sts : BOOL;
    RW_Pump_sts : BOOL;
    RW_Pump_fault : BOOL;
    RW_Pump : REAL;
    RW_Tank_PR_Valve : BOOL;
    RW_Tank_P_Valve : BOOL;
    RW_Pump_start : BOOL;
    RW_Pump_stop : BOOL;
    RW_Tank_P6B_Valve : BOOL;
  END_STRUCT;
  P2_UDT : STRUCT
    ChemTreat_NaCl_Tank_tnk_lvl : REAL;
    ChemTreat_NaOCl_Tank_tnk_lvl : REAL;
    ChemTreat_HCl_Tank_tnk_lvl : REAL;
    ChemTreat_NaCl_Tank_Valve_sts : BOOL;
    ChemTreat_NaOCl_Tank_Valve_sts : BOOL;
    ChemTreat_HCl_Tank_Valve_sts : BOOL;
    ChemTreat_NaCl_Tank_Valve : BOOL;
    ChemTreat_NaOCl_Tank_Valve : BOOL;
    ChemTreat_HCl_Tank_Valve : BOOL;
  END_STRUCT;
  P3_UDT : STRUCT
    Ultrafiltration_UFFT_Tank_tnk_lvl : REAL;
    Ultrafiltration_UFFT_Tank_Valve_sts : BOOL;
    Ultrafiltration_UF_Drain_Valve_sts : BOOL;
    Ultrafiltration_UF_ROFT_Valve_sts : BOOL;
    Ultrafiltration_UF_BWP_Valve_sts : BOOL;
    Ultrafiltration_UFFT_Tank_Valve : BOOL;
    Ultrafiltration_UF_Drain_Valve : BOOL;
    Ultrafiltration_UF_ROFT_Valve : BOOL;
    Ultrafiltration_UF_BWP_Valve : BOOL;
  END_STRUCT;
  Phases_UDT : STRUCT
    Filling : BOOL;
    Draining : BOOL;
  END_STRUCT;
  RW_tank_AL_UDT : STRUCT
    LL_alarm : BOOL;
    L_alarm : BOOL;
    H_alarm : BOOL;
    HH_alarm : BOOL;
  END_STRUCT;
  System_State_UDT : STRUCT
    IDLE : BOOL;
    START : BOOL;
    RUNNING : BOOL;
    SHUTDOWN : BOOL;
    Permissives : ARRAY [0..31] OF BOOL;
    Permissives_Ready : BOOL;
  END_STRUCT;
  SYS_MESSAGES : STRUCT
    ProgramScanTime : DINT;
    AvailableMemory : REAL;
    ControllerStatus : SINT;
    ScanTime : REAL;
  END_STRUCT;
END_TYPE

PROGRAM MainProgram
  VAR_INPUT
    Alarms : RW_tank_AL_UDT;
    GSV_Message : SYS_MESSAGES;
    P1 : P1_UDT;
    P1_SYS : System_State_UDT;
    P2 : P2_UDT;
    P3 : P3_UDT;
  END_VAR
  VAR_EXTERNAL
    di_2_0 : BOOL;
    di_2_1 : BOOL;
    di_2_10 : BOOL;
    di_2_11 : BOOL;
    di_2_2 : BOOL;
    di_2_3 : BOOL;
    di_2_4 : BOOL;
    di_2_5 : BOOL;
    di_2_6 : BOOL;
    di_2_8 : BOOL;
    di_2_9 : BOOL;
    ai_7_0 : REAL;
    di_7_ch0halarm : BOOL;
    di_7_ch0hhalarm : BOOL;
    di_7_ch0lalarm : BOOL;
    di_7_ch0llalarm : BOOL;
    ai_7_1 : REAL;
    ai_7_2 : REAL;
    ai_7_3 : REAL;
    ai_7_4 : REAL;
    ai_7_5 : REAL;
  END_VAR
  VAR_OUTPUT
    HMI : HMI_UDT;
  END_VAR
  VAR_EXTERNAL
    ao_10_0 : REAL;
    do_5_0 : BOOL;
    do_5_1 : BOOL;
    do_5_10 : BOOL;
    do_5_11 : BOOL;
    do_5_2 : BOOL;
    do_5_3 : BOOL;
    do_5_4 : BOOL;
    do_5_5 : BOOL;
    do_5_6 : BOOL;
    do_5_7 : BOOL;
    do_5_8 : BOOL;
    do_5_9 : BOOL;
  END_VAR

  (* IO_setup *)
  (* P1 Analog Input *)
  P1.RW_Tank_tnk_lvl := ai_7_0;
  P1.RW_Pump_flow := ai_7_1;
  (* P1 Digital Input *)
  P1.RW_Tank_PR_Valve_sts := di_2_0;
  P1.RW_Tank_P6B_Valve_sts := di_2_1;
  P1.RW_Tank_P_Valve_sts := di_2_2;
  P1.RW_Pump_sts := di_2_3;
  P1.RW_Pump_fault := di_2_4;
  (* P1 Analog Output *)
  P1.RW_Pump := ao_10_0;
  (* Digital Output *)
  P1.RW_Tank_PR_Valve := do_5_0;
  P1.RW_Tank_P6B_Valve := do_5_1;
  P1.RW_Tank_P_Valve := do_5_2;
  P1.RW_Pump_start := do_5_3;
  P1.RW_Pump_stop := do_5_4;
  (* P1 raw water tank alarms *)
  Alarms.LL_alarm := di_7_ch0llalarm;
  Alarms.L_alarm := di_7_ch0lalarm;
  Alarms.H_alarm := di_7_ch0halarm;
  Alarms.HH_alarm := di_7_ch0hhalarm;
  (* P2 Analog Input *)
  P2.ChemTreat_NaCl_Tank_tnk_lvl := ai_7_2;
  P2.ChemTreat_NaOCl_Tank_tnk_lvl := ai_7_3;
  P2.ChemTreat_HCl_Tank_tnk_lvl := ai_7_4;
  (* P2 Digital Input *)
  P2.ChemTreat_NaCl_Tank_Valve_sts := di_2_5;
  P2.ChemTreat_NaOCl_Tank_Valve_sts := di_2_6;
  (* P2 Analog Output *)
  (* NONE *)
  (* P2 Digital Output *)
  P2.ChemTreat_NaCl_Tank_Valve := do_5_5;
  P2.ChemTreat_NaOCl_Tank_Valve := do_5_6;
  P2.ChemTreat_HCl_Tank_Valve := do_5_7;
  (* P3 Analog Input *)
  P3.Ultrafiltration_UFFT_Tank_tnk_lvl := ai_7_5;
  (* P3 Digital Input *)
  P3.Ultrafiltration_UFFT_Tank_Valve_sts := di_2_8;
  P3.Ultrafiltration_UF_Drain_Valve_sts := di_2_9;
  P3.Ultrafiltration_UF_Drain_Valve_sts := di_2_10;
  P3.Ultrafiltration_UF_BWP_Valve_sts := di_2_11;
  (* P3 Analog Output *)
  (* none *)
  (* P3 Digital Output *)
  P3.Ultrafiltration_UFFT_Tank_Valve := do_5_8;
  P3.Ultrafiltration_UF_Drain_Valve := do_5_9;
  P3.Ultrafiltration_UF_ROFT_Valve := do_5_10;
  P3.Ultrafiltration_UF_BWP_Valve := do_5_11;

  (* Raw_water_control *)
  if P1.RW_Tank_tnk_lvl = 250.0 and P1_SYS.RUNNING then
  P1.RW_Pump_stop := True;
  P1.RW_Pump_start := False; (* send the outputs *)
  Alarms.LL_alarm := True;
  (* if the level is at 500 or lower than 500 open the valve *)
  elsif P1.RW_Tank_tnk_lvl <= 500.0 and P1_SYS.RUNNING then
  (* output to turn the valve open *)
  P1.RW_Tank_PR_Valve := True;
  Alarms.L_alarm := True;
  (* if level is at 800 *)
  elsif  P1.RW_Tank_tnk_lvl = 800.0 and P1_SYS.RUNNING then
  P1.RW_Tank_PR_Valve := False; (* close the valve *)
  Alarms.H_alarm := True;
  elsif P1.RW_Tank_tnk_lvl = 1200.0 and P1_SYS.RUNNING then
  Alarms.HH_alarm := True; (* if the tank is higher than or equal to 1200 set the high high alarm *)
  end_if;

  (* Raw_water_pump *)
  if P3.Ultrafiltration_UFFT_Tank_tnk_lvl = 800.0 AND P1_SYS.RUNNING then
  (* start the pump and open the valve from the other tank *)
  P1.RW_Tank_P_Valve := True;
  P1.RW_Pump_start := True;
  P1.RW_Pump_stop := False;
  elsif P3.Ultrafiltration_UFFT_Tank_tnk_lvl = 1000.0 AND P1_SYS.RUNNING then
  (* stop the pump and close the valve *)
  P1.RW_Tank_P_Valve := False;
  P1.RW_Pump_stop := True;
  P1.RW_Pump_start := False;
  end_if;

  (* State_change *)
  if not HMI.Start_Active AND not HMI.Stop_Active then
  (* if start and stop is not pressed go to idle *)
  P1_SYS.IDLE := True;
  P1_SYS.START := False;
  P1_SYS.RUNNING := False;
  P1_SYS.SHUTDOWN := False;
  elsif  HMI.Start_Active AND not HMI.Stop_Active then
  (* if the start pb and stop is not pressed then change the state of process one to starting *)
  P1_SYS.IDLE := False;
  P1_SYS.START := True;
  P1_SYS.RUNNING := False;
  P1_SYS.SHUTDOWN := False;
  (* if the tank level is greater than 250 at the start and UFFT is less than a 1000 we can start *)
  (* then and all permissves cond together into one tag so we know the plant is ready to start *)
  P1_SYS.Permissives_Ready := P1_SYS.Permissives[0] AND P1_SYS.Permissives[1];
  elsif HMI.Start_Active AND P1_SYS.Permissives_Ready then
  (* if the start was pressed and permissives are ready start running Process one *)
  P1_SYS.IDLE := False;
  P1_SYS.START := False;
  P1_SYS.RUNNING := True;
  P1_SYS.SHUTDOWN := False;
  elsif HMI.Stop_Active then
  (* if the stop button is pressed then go to shutdown state *)
  P1_SYS.IDLE := False;
  P1_SYS.START := False;
  P1_SYS.RUNNING := False;
  P1_SYS.SHUTDOWN := True;
  (* set all permissives to false *)
  P1_SYS.Permissives_Ready := False;
  end_if;
END_PROGRAM

CONFIGURATION config
  VAR_GLOBAL
    ao_10_0 AT %QW100 : REAL;
    di_2_0 AT %IX2.0 : BOOL;
    di_2_1 AT %IX2.1 : BOOL;
    di_2_10 AT %IX2.10 : BOOL;
    di_2_11 AT %IX2.11 : BOOL;
    di_2_2 AT %IX2.2 : BOOL;
    di_2_3 AT %IX2.3 : BOOL;
    di_2_4 AT %IX2.4 : BOOL;
    di_2_5 AT %IX2.5 : BOOL;
    di_2_6 AT %IX2.6 : BOOL;
    di_2_8 AT %IX2.8 : BOOL;
    di_2_9 AT %IX2.9 : BOOL;
    do_5_0 AT %QX5.0 : BOOL;
    do_5_1 AT %QX5.1 : BOOL;
    do_5_10 AT %QX5.10 : BOOL;
    do_5_11 AT %QX5.11 : BOOL;
    do_5_2 AT %QX5.2 : BOOL;
    do_5_3 AT %QX5.3 : BOOL;
    do_5_4 AT %QX5.4 : BOOL;
    do_5_5 AT %QX5.5 : BOOL;
    do_5_6 AT %QX5.6 : BOOL;
    do_5_7 AT %QX5.7 : BOOL;
    do_5_8 AT %QX5.8 : BOOL;
    do_5_9 AT %QX5.9 : BOOL;
    ai_7_0 AT %IW70 : REAL;
    di_7_ch0halarm AT %IX7.0 : BOOL;
    di_7_ch0hhalarm AT %IX7.0 : BOOL;
    di_7_ch0lalarm AT %IX7.0 : BOOL;
    di_7_ch0llalarm AT %IX7.0 : BOOL;
    ai_7_1 AT %IW71 : REAL;
    ai_7_2 AT %IW72 : REAL;
    ai_7_3 AT %IW73 : REAL;
    ai_7_4 AT %IW74 : REAL;
    ai_7_5 AT %IW75 : REAL;
  END_VAR

  RESOURCE res_MainProgram ON PLC
    TASK task_MainProgram(INTERVAL := T#100ms,PRIORITY := 0);
    PROGRAM MainProgram_instance : MainProgram;
  END_RESOURCE
END_CONFIGURATION

(*DBG:char md5[] = "527971c67af0de80c69f5223004ec189";*)
(*DBG:/**)
(*DBG: * This file is part of OpenPLC Runtime*)
(*DBG: **)
(*DBG: * Copyright (C) 2023 Autonomy, GP Orcullo*)
(*DBG: * Based on the work by GP Orcullo on Beremiz for uC*)
(*DBG: **)
(*DBG: * This program is free software; you can redistribute it and/or*)
(*DBG: * modify it under the terms of the GNU General Public License*)
(*DBG: * as published by the Free Software Foundation; either version 2*)
(*DBG: * of the License, or (at your option) any later version.*)
(*DBG: **)
(*DBG: * This program is distributed in the hope that it will be useful,*)
(*DBG: * but WITHOUT ANY WARRANTY; without even the implied warranty of*)
(*DBG: * MERCHANTABILITY or FITNESS FOR A PARTICULAR PURPOSE.  See the*)
(*DBG: * GNU General Public License for more details.*)
(*DBG: **)
(*DBG: * You should have received a copy of the GNU General Public License*)
(*DBG: * along with this program; If not, see <http://www.gnu.org/licenses/>.*)
(*DBG: **)
(*DBG: */*)
(*DBG:*)
(*DBG:#include <stdbool.h>*)
(*DBG:*)
(*DBG:#include "iec_types_all.h"*)
(*DBG:#include "POUS.h"*)
(*DBG:*)
(*DBG:#define SAME_ENDIANNESS      0*)
(*DBG:#define REVERSE_ENDIANNESS   1*)
(*DBG:*)
(*DBG:uint8_t endianness;*)
(*DBG:*)
(*DBG:*)
(*DBG:extern __IEC_REAL_t CONFIG__AO_10_0;*)
(*DBG:extern __IEC_BOOL_t CONFIG__DI_2_0;*)
(*DBG:extern __IEC_BOOL_t CONFIG__DI_2_1;*)
(*DBG:extern __IEC_BOOL_t CONFIG__DI_2_10;*)
(*DBG:extern __IEC_BOOL_t CONFIG__DI_2_11;*)
(*DBG:extern __IEC_BOOL_t CONFIG__DI_2_2;*)
(*DBG:extern __IEC_BOOL_t CONFIG__DI_2_3;*)
(*DBG:extern __IEC_BOOL_t CONFIG__DI_2_4;*)
(*DBG:extern __IEC_BOOL_t CONFIG__DI_2_5;*)
(*DBG:extern __IEC_BOOL_t CONFIG__DI_2_6;*)
(*DBG:extern __IEC_BOOL_t CONFIG__DI_2_8;*)
(*DBG:extern __IEC_BOOL_t CONFIG__DI_2_9;*)
(*DBG:extern __IEC_BOOL_t CONFIG__DO_5_0;*)
(*DBG:extern __IEC_BOOL_t CONFIG__DO_5_1;*)
(*DBG:extern __IEC_BOOL_t CONFIG__DO_5_10;*)
(*DBG:extern __IEC_BOOL_t CONFIG__DO_5_11;*)
(*DBG:extern __IEC_BOOL_t CONFIG__DO_5_2;*)
(*DBG:extern __IEC_BOOL_t CONFIG__DO_5_3;*)
(*DBG:extern __IEC_BOOL_t CONFIG__DO_5_4;*)
(*DBG:extern __IEC_BOOL_t CONFIG__DO_5_5;*)
(*DBG:extern __IEC_BOOL_t CONFIG__DO_5_6;*)
(*DBG:extern __IEC_BOOL_t CONFIG__DO_5_7;*)
(*DBG:extern __IEC_BOOL_t CONFIG__DO_5_8;*)
(*DBG:extern __IEC_BOOL_t CONFIG__DO_5_9;*)
(*DBG:extern __IEC_REAL_t CONFIG__AI_7_0;*)
(*DBG:extern __IEC_BOOL_t CONFIG__DI_7_CH0HALARM;*)
(*DBG:extern __IEC_BOOL_t CONFIG__DI_7_CH0HHALARM;*)
(*DBG:extern __IEC_BOOL_t CONFIG__DI_7_CH0LALARM;*)
(*DBG:extern __IEC_BOOL_t CONFIG__DI_7_CH0LLALARM;*)
(*DBG:extern __IEC_REAL_t CONFIG__AI_7_1;*)
(*DBG:extern __IEC_REAL_t CONFIG__AI_7_2;*)
(*DBG:extern __IEC_REAL_t CONFIG__AI_7_3;*)
(*DBG:extern __IEC_REAL_t CONFIG__AI_7_4;*)
(*DBG:extern __IEC_REAL_t CONFIG__AI_7_5;*)
(*DBG:extern MAINPROGRAM RES_MAINPROGRAM__MAINPROGRAM_INSTANCE;*)
(*DBG:*)
(*DBG:static const struct {*)
(*DBG:    void *ptr;*)
(*DBG:    __IEC_types_enum type;*)
(*DBG:} debug_vars[] = {*)
(*DBG:    {&(CONFIG__AO_10_0), REAL_ENUM},*)
(*DBG:    {&(CONFIG__DI_2_0), BOOL_ENUM},*)
(*DBG:    {&(CONFIG__DI_2_1), BOOL_ENUM},*)
(*DBG:    {&(CONFIG__DI_2_10), BOOL_ENUM},*)
(*DBG:    {&(CONFIG__DI_2_11), BOOL_ENUM},*)
(*DBG:    {&(CONFIG__DI_2_2), BOOL_ENUM},*)
(*DBG:    {&(CONFIG__DI_2_3), BOOL_ENUM},*)
(*DBG:    {&(CONFIG__DI_2_4), BOOL_ENUM},*)
(*DBG:    {&(CONFIG__DI_2_5), BOOL_ENUM},*)
(*DBG:    {&(CONFIG__DI_2_6), BOOL_ENUM},*)
(*DBG:    {&(CONFIG__DI_2_8), BOOL_ENUM},*)
(*DBG:    {&(CONFIG__DI_2_9), BOOL_ENUM},*)
(*DBG:    {&(CONFIG__DO_5_0), BOOL_ENUM},*)
(*DBG:    {&(CONFIG__DO_5_1), BOOL_ENUM},*)
(*DBG:    {&(CONFIG__DO_5_10), BOOL_ENUM},*)
(*DBG:    {&(CONFIG__DO_5_11), BOOL_ENUM},*)
(*DBG:    {&(CONFIG__DO_5_2), BOOL_ENUM},*)
(*DBG:    {&(CONFIG__DO_5_3), BOOL_ENUM},*)
(*DBG:    {&(CONFIG__DO_5_4), BOOL_ENUM},*)
(*DBG:    {&(CONFIG__DO_5_5), BOOL_ENUM},*)
(*DBG:    {&(CONFIG__DO_5_6), BOOL_ENUM},*)
(*DBG:    {&(CONFIG__DO_5_7), BOOL_ENUM},*)
(*DBG:    {&(CONFIG__DO_5_8), BOOL_ENUM},*)
(*DBG:    {&(CONFIG__DO_5_9), BOOL_ENUM},*)
(*DBG:    {&(CONFIG__AI_7_0), REAL_ENUM},*)
(*DBG:    {&(CONFIG__DI_7_CH0HALARM), BOOL_ENUM},*)
(*DBG:    {&(CONFIG__DI_7_CH0HHALARM), BOOL_ENUM},*)
(*DBG:    {&(CONFIG__DI_7_CH0LALARM), BOOL_ENUM},*)
(*DBG:    {&(CONFIG__DI_7_CH0LLALARM), BOOL_ENUM},*)
(*DBG:    {&(CONFIG__AI_7_1), REAL_ENUM},*)
(*DBG:    {&(CONFIG__AI_7_2), REAL_ENUM},*)
(*DBG:    {&(CONFIG__AI_7_3), REAL_ENUM},*)
(*DBG:    {&(CONFIG__AI_7_4), REAL_ENUM},*)
(*DBG:    {&(CONFIG__AI_7_5), REAL_ENUM},*)
(*DBG:    {&(RES_MAINPROGRAM__MAINPROGRAM_INSTANCE.DI_2_0), BOOL_ENUM},*)
(*DBG:    {&(RES_MAINPROGRAM__MAINPROGRAM_INSTANCE.DI_2_1), BOOL_ENUM},*)
(*DBG:    {&(RES_MAINPROGRAM__MAINPROGRAM_INSTANCE.DI_2_10), BOOL_ENUM},*)
(*DBG:    {&(RES_MAINPROGRAM__MAINPROGRAM_INSTANCE.DI_2_11), BOOL_ENUM},*)
(*DBG:    {&(RES_MAINPROGRAM__MAINPROGRAM_INSTANCE.DI_2_2), BOOL_ENUM},*)
(*DBG:    {&(RES_MAINPROGRAM__MAINPROGRAM_INSTANCE.DI_2_3), BOOL_ENUM},*)
(*DBG:    {&(RES_MAINPROGRAM__MAINPROGRAM_INSTANCE.DI_2_4), BOOL_ENUM},*)
(*DBG:    {&(RES_MAINPROGRAM__MAINPROGRAM_INSTANCE.DI_2_5), BOOL_ENUM},*)
(*DBG:    {&(RES_MAINPROGRAM__MAINPROGRAM_INSTANCE.DI_2_6), BOOL_ENUM},*)
(*DBG:    {&(RES_MAINPROGRAM__MAINPROGRAM_INSTANCE.DI_2_8), BOOL_ENUM},*)
(*DBG:    {&(RES_MAINPROGRAM__MAINPROGRAM_INSTANCE.DI_2_9), BOOL_ENUM},*)
(*DBG:    {&(RES_MAINPROGRAM__MAINPROGRAM_INSTANCE.AI_7_0), REAL_ENUM},*)
(*DBG:    {&(RES_MAINPROGRAM__MAINPROGRAM_INSTANCE.DI_7_CH0HALARM), BOOL_ENUM},*)
(*DBG:    {&(RES_MAINPROGRAM__MAINPROGRAM_INSTANCE.DI_7_CH0HHALARM), BOOL_ENUM},*)
(*DBG:    {&(RES_MAINPROGRAM__MAINPROGRAM_INSTANCE.DI_7_CH0LALARM), BOOL_ENUM},*)
(*DBG:    {&(RES_MAINPROGRAM__MAINPROGRAM_INSTANCE.DI_7_CH0LLALARM), BOOL_ENUM},*)
(*DBG:    {&(RES_MAINPROGRAM__MAINPROGRAM_INSTANCE.AI_7_1), REAL_ENUM},*)
(*DBG:    {&(RES_MAINPROGRAM__MAINPROGRAM_INSTANCE.AI_7_2), REAL_ENUM},*)
(*DBG:    {&(RES_MAINPROGRAM__MAINPROGRAM_INSTANCE.AI_7_3), REAL_ENUM},*)
(*DBG:    {&(RES_MAINPROGRAM__MAINPROGRAM_INSTANCE.AI_7_4), REAL_ENUM},*)
(*DBG:    {&(RES_MAINPROGRAM__MAINPROGRAM_INSTANCE.AI_7_5), REAL_ENUM},*)
(*DBG:    {&(RES_MAINPROGRAM__MAINPROGRAM_INSTANCE.AO_10_0), REAL_ENUM},*)
(*DBG:    {&(RES_MAINPROGRAM__MAINPROGRAM_INSTANCE.DO_5_0), BOOL_ENUM},*)
(*DBG:    {&(RES_MAINPROGRAM__MAINPROGRAM_INSTANCE.DO_5_1), BOOL_ENUM},*)
(*DBG:    {&(RES_MAINPROGRAM__MAINPROGRAM_INSTANCE.DO_5_10), BOOL_ENUM},*)
(*DBG:    {&(RES_MAINPROGRAM__MAINPROGRAM_INSTANCE.DO_5_11), BOOL_ENUM},*)
(*DBG:    {&(RES_MAINPROGRAM__MAINPROGRAM_INSTANCE.DO_5_2), BOOL_ENUM},*)
(*DBG:    {&(RES_MAINPROGRAM__MAINPROGRAM_INSTANCE.DO_5_3), BOOL_ENUM},*)
(*DBG:    {&(RES_MAINPROGRAM__MAINPROGRAM_INSTANCE.DO_5_4), BOOL_ENUM},*)
(*DBG:    {&(RES_MAINPROGRAM__MAINPROGRAM_INSTANCE.DO_5_5), BOOL_ENUM},*)
(*DBG:    {&(RES_MAINPROGRAM__MAINPROGRAM_INSTANCE.DO_5_6), BOOL_ENUM},*)
(*DBG:    {&(RES_MAINPROGRAM__MAINPROGRAM_INSTANCE.DO_5_7), BOOL_ENUM},*)
(*DBG:    {&(RES_MAINPROGRAM__MAINPROGRAM_INSTANCE.DO_5_8), BOOL_ENUM},*)
(*DBG:    {&(RES_MAINPROGRAM__MAINPROGRAM_INSTANCE.DO_5_9), BOOL_ENUM},*)
(*DBG:};*)
(*DBG:*)
(*DBG:#define VAR_COUNT               68*)
(*DBG:*)
(*DBG:uint16_t get_var_count(void)*)
(*DBG:{*)
(*DBG:    return VAR_COUNT;*)
(*DBG:}*)
(*DBG:*)
(*DBG:size_t get_var_size(size_t idx)*)
(*DBG:{*)
(*DBG:    if (idx >= VAR_COUNT)*)
(*DBG:    {*)
(*DBG:        return 0;*)
(*DBG:    }*)
(*DBG:    switch (debug_vars[idx].type) {*)
(*DBG:    case REAL_ENUM:*)
(*DBG:        return sizeof(REAL);*)
(*DBG:    case BOOL_ENUM:*)
(*DBG:        return sizeof(BOOL);*)
(*DBG:    default:*)
(*DBG:        return 0;*)
(*DBG:    }*)
(*DBG:}*)
(*DBG:*)
(*DBG:void *get_var_addr(size_t idx)*)
(*DBG:{*)
(*DBG:    void *ptr = debug_vars[idx].ptr;*)
(*DBG:*)
(*DBG:    switch (debug_vars[idx].type) {*)
(*DBG:    case REAL_ENUM:*)
(*DBG:        return (void *)&((__IEC_REAL_t *) ptr)->value;*)
(*DBG:    case BOOL_ENUM:*)
(*DBG:        return (void *)&((__IEC_BOOL_t *) ptr)->value;*)
(*DBG:    default:*)
(*DBG:        return 0;*)
(*DBG:    }*)
(*DBG:}*)
(*DBG:*)
(*DBG:void force_var(size_t idx, bool forced, void *val)*)
(*DBG:{*)
(*DBG:    void *ptr = debug_vars[idx].ptr;*)
(*DBG:*)
(*DBG:    if (forced) {*)
(*DBG:        size_t var_size = get_var_size(idx);*)
(*DBG:        switch (debug_vars[idx].type) {*)
(*DBG:        case REAL_ENUM: {*)
(*DBG:            memcpy(&((__IEC_REAL_t *) ptr)->value, val, var_size);*)
(*DBG:            //((__IEC_REAL_t *) ptr)->value = *((REAL *) val);*)
(*DBG:            ((__IEC_REAL_t *) ptr)->flags |= __IEC_FORCE_FLAG;*)
(*DBG:            break;*)
(*DBG:        }*)
(*DBG:        case BOOL_ENUM: {*)
(*DBG:            memcpy(&((__IEC_BOOL_t *) ptr)->value, val, var_size);*)
(*DBG:            //((__IEC_BOOL_t *) ptr)->value = *((BOOL *) val);*)
(*DBG:            ((__IEC_BOOL_t *) ptr)->flags |= __IEC_FORCE_FLAG;*)
(*DBG:            break;*)
(*DBG:        }*)
(*DBG:        default:*)
(*DBG:            break;*)
(*DBG:        }*)
(*DBG:    } else {*)
(*DBG:        switch (debug_vars[idx].type) {*)
(*DBG:        case REAL_ENUM:*)
(*DBG:            ((__IEC_REAL_t *) ptr)->flags &= ~__IEC_FORCE_FLAG;*)
(*DBG:            break;*)
(*DBG:        case BOOL_ENUM:*)
(*DBG:            ((__IEC_BOOL_t *) ptr)->flags &= ~__IEC_FORCE_FLAG;*)
(*DBG:            break;*)
(*DBG:        default:*)
(*DBG:            break;*)
(*DBG:        }*)
(*DBG:    }*)
(*DBG:}*)
(*DBG:*)
(*DBG:void swap_bytes(void *ptr, size_t size) *)
(*DBG:{*)
(*DBG:    uint8_t *bytePtr = (uint8_t *)ptr;*)
(*DBG:    size_t i;*)
(*DBG:    for (i = 0; i < size / 2; ++i) *)
(*DBG:    {*)
(*DBG:        uint8_t temp = bytePtr[i];*)
(*DBG:        bytePtr[i] = bytePtr[size - 1 - i];*)
(*DBG:        bytePtr[size - 1 - i] = temp;*)
(*DBG:    }*)
(*DBG:}*)
(*DBG:*)
(*DBG:void trace_reset(void)*)
(*DBG:{*)
(*DBG:    for (size_t i=0; i < VAR_COUNT; i++) *)
(*DBG:    {*)
(*DBG:        force_var(i, false, 0);*)
(*DBG:    }*)
(*DBG:}*)
(*DBG:*)
(*DBG:void set_trace(size_t idx, bool forced, void *val)*)
(*DBG:{*)
(*DBG:    if (idx >= 0 && idx < VAR_COUNT) *)
(*DBG:    {*)
(*DBG:        if (endianness == REVERSE_ENDIANNESS)*)
(*DBG:        {*)
(*DBG:            // Aaaaarghhhh... Stupid AVR is Big Endian.*)
(*DBG:            swap_bytes(val, get_var_size(idx));*)
(*DBG:        }*)
(*DBG:*)
(*DBG:        force_var(idx, forced, val);*)
(*DBG:    }*)
(*DBG:}*)
(*DBG:*)
(*DBG:void set_endianness(uint8_t value)*)
(*DBG:{*)
(*DBG:    if (value == SAME_ENDIANNESS || value == REVERSE_ENDIANNESS)*)
(*DBG:    {*)
(*DBG:        endianness = value;*)
(*DBG:    }*)
(*DBG:}*)
(*DBG:*)
